FUNCTION_BLOCK SH_1
VAR_INPUT
	in : REAL;
	PT : TIME;
END_VAR
VAR_OUTPUT
	out : REAL;
	Trig : BOOL;
END_VAR
VAR
	last : TIME;
	tx: TIME;
END_VAR

(*
version 1.2	17 sep 2007
programmer 	hugo
tested by		tobias

this sample and hold module samples an input every PT seconds.
after a ample is taken the output Trig will be active for one cycle.

*)

(* read system time *)
tx := DWORD_TO_TIME(T_PLC_MS());

IF tx - last >= PT THEN
	last := tx;
	out := in;
	trig := TRUE;
ELSE
	trig := FALSE;
END_IF;

(* revision history

HM	6.1.2007	rev 1.1
	added trig output

HM	17.9.2007	rev 1.2
	replaced time() with T_PLC_MS() for compatibility reasons
*)

END_FUNCTION_BLOCK

(* stored: Version 1.1.0.1, ProductVersion 3.1.4022.7
   POU SH_1: Id {22f7c3c9-2fc9-4d9d-ae94-aab82132aeb0}, SpecialFunc None *)
